// TwinCAT 3 PLC project Motor_1DK
// ProgramVersion: 3.1.4024.0
// libraries:
//   Tc2_Standard, * (Beckhoff Automation GmbH)
//   Tc2_System, * (Beckhoff Automation GmbH)
//   Tc3_Module, * (Beckhoff Automation GmbH)
// project tree:
//   / PlcTask.TcTTO
//   POUs/ MAIN.TcPOU

CONFIGURATION Motor_1DK
    RESOURCE PLC ON TwinCAT3
        TASK PlcTask(INTERVAL := T#10ms, PRIORITY := 27);
        PROGRAM MAIN WITH PlcTask : MAIN;
    END_RESOURCE
END_CONFIGURATION

// ---- POUs/MAIN.TcPOU
PROGRAM MAIN
VAR
	
// Inputs
	HoofdSchakelaar: BOOL;
	prevDrukKnop: BOOL;
	DrukKnop: BOOL;
	Teller: INT;

// Outputs
	MotorLinks: BOOL;
	MotorRechts: BOOL;

END_VAR

(*
Motor starten met één drukknop (4 regels code)

Schrijf een programma om een motor [ Relais voor MotorLinks en MotorRechts ] te starten en te stoppen met één drukknop. 
De installatie zal pas werken als een hoofdschakelaar AAN staat.

    1e druk op de drukknop:	start links draaiend
    2e druk op de drukknop:	stop
    3e druk op de drukknop:	start rechts draaiend
    4e druk op de drukknop:	stop
*)

IF HoofdSchakelaar AND NOT prevDrukKnop AND DrukKnop THEN Teller := (Teller + 1) MOD 4; END_IF;
prevDrukKnop := DrukKnop;
MotorLinks := HoofdSchakelaar AND Teller = 1;
MotorRechts := HoofdSchakelaar AND Teller = 3;

END_PROGRAM
